// TwinCAT 3 PLC project PLCserra
// ProgramVersion: 3.1.4024.0
// libraries:
//   Tc2_Standard, * (Beckhoff Automation GmbH)
//   Tc2_System, * (Beckhoff Automation GmbH)
//   Tc3_Module, * (Beckhoff Automation GmbH)
// project tree:
//   / PlcTask.TcTTO (not stored)
//   POUs/ main.TcPOU
// real-time tasks:
//   TASK PlcTask: cycle T#10ms, priority 20, ADS port 350

// ---- POUs/main.TcPOU
PROGRAM main
VAR
	//attuatori
	AttuatBraccioGiu : BOOL := FALSE;
	AttuatBraccioSu : BOOL := FALSE;
	AttuatBraccioSx : BOOL := FALSE;
	AttuatBraccioDx : BOOL := FALSE;
	AttuatBraccioPresa : BOOL := FALSE;
	AttuatBraccioRilascio : BOOL := FALSE;
	AttuatRiempiSerbatoio : BOOL := FALSE;
	AttuatSvuotaSerbatoio : BOOL := FALSE;
	AttuatFinestra : BOOL := FALSE;
	AttuatCondizionatore : BOOL := FALSE;
	AttuatRullo : BOOL := FALSE;
	AttuatLampada : BOOL := FALSE;
	//sensori
	SensoreFCB : BOOL := FALSE;
	SensoreFCT : BOOL := FALSE;
	SensoreFCS : BOOL := FALSE;
	SensoreFCD : BOOL := FALSE;
	SensoreFineCorsaPianta2 : BOOL := FALSE;
	SensoreGrasp : BOOL := FALSE;
	SensoreRelease : BOOL := FALSE;
	SensoreRulloOccupato : BOOL := FALSE;
	SensoreVascaPienaVuota : BOOL := FALSE;
	SensoreSerbatoioOn : BOOL := FALSE;
	SensoreSerbatoioFull : BOOL := FALSE;
	SensoreSerbatoioEmpty : BOOL := FALSE;
	SensoreCondizionatore : BOOL := FALSE;
	SensoreLuci : BOOL := FALSE;
	SensoreFinestra : BOOL := FALSE;
	SensoreTempCalda : BOOL := FALSE;
	SensoreTempFredda : BOOL := FALSE;
	SensorePianta1Pronta : BOOL := FALSE;
	SensorePianta2Pronta : BOOL := FALSE;
	SensoreStart : BOOL := FALSE;
	SensoreReset : BOOL := FALSE;
	//Variabili Controllo temperatura
	TemperaturaAttuale : INT;
	TemperaturaOttimale : INT := 36;
	
	//Variabili Controllo luce
	durataGiorno : INT;
	durataNotte : INT;
	
	//Variabili controllo Serbatoio
	LivelloSerbatoio : INT;
	LivelloSerbatoioMax : INT;
	
	
	SerbatoioVuoto: BOOL;
	Pianta1Pronta: INT;
	SerbatoioPieno: BOOL;
	VascaVuota: BOOL;
	VascaPiena: BOOL;
	Pianta2Pronta: BOOL;
	RulloPieno: BOOL;
	SopraPianta1: INT;
	PrendiPianta1: BOOL;
	PosizionePianta1: BOOL;
	Pianta1Grasped: BOOL;
	Pianta1Sopra: BOOL;
	Pianta1Alzata: BOOL;
	Pianta1SopraRullo: BOOL;
	Pianta1SulRullo: INT;
	SulRullo: INT;
	Pianta1SulRulloSulRullo: BOOL;
	Pianta1Rilasciata: BOOL;
	SopraPianta2: INT;
END_VAR

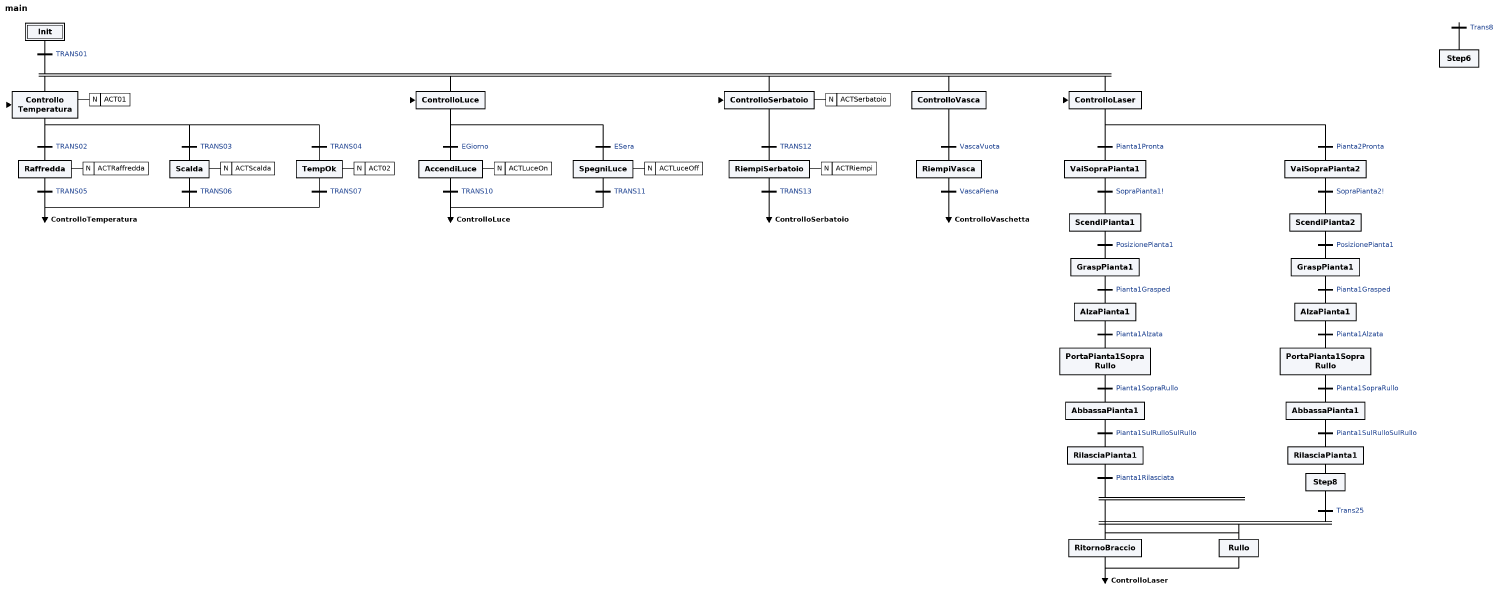
INITIAL_STEP Init:
END_STEP
TRANSITION FROM Init TO (ControlloTemperatura, ControlloLuce, ControlloSerbatoio, ControlloVasca, ControlloLaser)
    := TRANS01;
END_TRANSITION
STEP ControlloTemperatura:
    ACT01(N);
END_STEP
TRANSITION FROM ControlloTemperatura TO Raffredda
    := TRANS02;
END_TRANSITION
STEP Raffredda:
    ACTRaffredda(N);
END_STEP
TRANSITION FROM Raffredda TO ControlloTemperatura
    := TRANS05;
END_TRANSITION
TRANSITION FROM ControlloTemperatura TO Scalda
    := TRANS03;
END_TRANSITION
STEP Scalda:
    ACTScalda(N);
END_STEP
TRANSITION FROM Scalda TO ControlloTemperatura
    := TRANS06;
END_TRANSITION
TRANSITION FROM ControlloTemperatura TO TempOk
    := TRANS04;
END_TRANSITION
STEP TempOk:
    ACT02(N);
END_STEP
TRANSITION FROM TempOk TO ControlloTemperatura
    := TRANS07;
END_TRANSITION
STEP ControlloLuce:
END_STEP
TRANSITION FROM ControlloLuce TO AccendiLuce
    := EGiorno;
END_TRANSITION
STEP AccendiLuce:
    ACTLuceOn(N);
END_STEP
TRANSITION FROM AccendiLuce TO ControlloLuce
    := TRANS10;
END_TRANSITION
TRANSITION FROM ControlloLuce TO SpegniLuce
    := ESera;
END_TRANSITION
STEP SpegniLuce:
    ACTLuceOff(N);
END_STEP
TRANSITION FROM SpegniLuce TO ControlloLuce
    := TRANS11;
END_TRANSITION
STEP ControlloSerbatoio:
    ACTSerbatoio(N);
END_STEP
TRANSITION FROM ControlloSerbatoio TO RiempiSerbatoio
    := TRANS12;
END_TRANSITION
STEP RiempiSerbatoio:
    ACTRiempi(N);
END_STEP
TRANSITION FROM RiempiSerbatoio TO ControlloSerbatoio
    := TRANS13;
END_TRANSITION
STEP ControlloVasca:
END_STEP
TRANSITION FROM ControlloVasca TO RiempiVasca
    := VascaVuota;
END_TRANSITION
STEP RiempiVasca:
END_STEP
TRANSITION FROM RiempiVasca TO ControlloVaschetta
    := VascaPiena;
END_TRANSITION
STEP ControlloLaser:
END_STEP
TRANSITION FROM ControlloLaser TO VaiSopraPianta1
    := Pianta1Pronta;
END_TRANSITION
STEP VaiSopraPianta1:
END_STEP
TRANSITION FROM VaiSopraPianta1 TO ScendiPianta1
    := SopraPianta1!;
END_TRANSITION
STEP ScendiPianta1:
END_STEP
TRANSITION FROM ScendiPianta1 TO GraspPianta1
    := PosizionePianta1;
END_TRANSITION
STEP GraspPianta1:
END_STEP
TRANSITION FROM GraspPianta1 TO AlzaPianta1
    := Pianta1Grasped;
END_TRANSITION
STEP AlzaPianta1:
END_STEP
TRANSITION FROM AlzaPianta1 TO PortaPianta1SopraRullo
    := Pianta1Alzata;
END_TRANSITION
STEP PortaPianta1SopraRullo:
END_STEP
TRANSITION FROM PortaPianta1SopraRullo TO AbbassaPianta1
    := Pianta1SopraRullo;
END_TRANSITION
STEP AbbassaPianta1:
END_STEP
TRANSITION FROM AbbassaPianta1 TO RilasciaPianta1
    := Pianta1SulRulloSulRullo;
END_TRANSITION
STEP RilasciaPianta1:
END_STEP
TRANSITION FROM RilasciaPianta1 TO (RitornoBraccio, Rullo)
    := Pianta1Rilasciata;
END_TRANSITION
TRANSITION FROM ControlloLaser TO VaiSopraPianta2
    := Pianta2Pronta;
END_TRANSITION
STEP VaiSopraPianta2:
END_STEP
TRANSITION FROM VaiSopraPianta2 TO ScendiPianta2
    := SopraPianta2!;
END_TRANSITION
STEP ScendiPianta2:
END_STEP
TRANSITION FROM ScendiPianta2 TO GraspPianta1
    := PosizionePianta1;
END_TRANSITION
STEP GraspPianta1:
END_STEP
TRANSITION FROM GraspPianta1 TO AlzaPianta1
    := Pianta1Grasped;
END_TRANSITION
STEP AlzaPianta1:
END_STEP
TRANSITION FROM AlzaPianta1 TO PortaPianta1SopraRullo
    := Pianta1Alzata;
END_TRANSITION
STEP PortaPianta1SopraRullo:
END_STEP
TRANSITION FROM PortaPianta1SopraRullo TO AbbassaPianta1
    := Pianta1SopraRullo;
END_TRANSITION
STEP AbbassaPianta1:
END_STEP
TRANSITION FROM AbbassaPianta1 TO RilasciaPianta1
    := Pianta1SulRulloSulRullo;
END_TRANSITION
STEP RilasciaPianta1:
END_STEP
// no transition between RilasciaPianta1 and Step8
STEP Step8:
END_STEP
TRANSITION FROM Step8 TO (RitornoBraccio, Rullo)
    := Trans25;
END_TRANSITION
STEP RitornoBraccio:
END_STEP
// no transition between RitornoBraccio and ControlloLaser
STEP Rullo:
END_STEP
// no transition between Rullo and ControlloLaser
TRANSITION FROM ??? TO Step6
    := Trans8;
END_TRANSITION
STEP Step6:
END_STEP

ACTION ACT01:
IF TemperaturaAttuale < TemperaturaOttimale-5 THEN
	SensoreTempFredda := TRUE;
	SensoreTempCalda := FALSE;
	
ELSIF TemperaturaAttuale > TemperaturaOttimale+5 THEN
	SensoreTempCalda := TRUE;
	SensoreTempFredda := FALSE;
END_IF
END_ACTION

ACTION ACT02:
AttuatCondizionatore := FALSE;
END_ACTION

ACTION ACTLuceOff:
AttuatLampada := FALSE;
SensoreLuci := FALSE;
END_ACTION

ACTION ACTLuceOn:
AttuatLampada := TRUE;
SensoreLuci := TRUE;
END_ACTION

ACTION ACTRaffredda:
//Dovrebbe azionare il condizionare freddo
AttuatCondizionatore := TRUE;
END_ACTION

ACTION ACTRiempi:
AttuatRiempiSerbatoio := TRUE;
SensoreSerbatoioEmpty := FALSE;
END_ACTION

ACTION ACTScalda:
//Dovrebbe azionare il condizionatore caldo
AttuatCondizionatore := TRUE;
END_ACTION

ACTION ACTSerbatoio:
IF LivelloSerbatoio > 0 THEN
	IF LivelloSerbatoio = LivelloSerbatoioMax THEN
		SensoreSerbatoioFull := TRUE;
		SensoreSerbatoioEmpty := FALSE;
	END_IF
	SensoreSerbatoioEmpty := FALSE;
END_IF

IF LivelloSerbatoio = 0 THEN
	SensoreSerbatoioEmpty := TRUE;
	SensoreSerbatoioFull := FALSE;
	AttuatRiempiSerbatoio := TRUE;
END_IF
END_ACTION

TRANSITION TRANS01:
SensoreStart = TRUE AND SensoreFCTop= TRUE AND SensoreFCD = TRUE AND SensoreRulloOccupato = FALSE;
END_TRANSITION

TRANSITION TRANS02:
SensoreTempCalda := TRUE;
END_TRANSITION

TRANSITION TRANS03:
SensoreTempFredda := TRUE;
END_TRANSITION

TRANSITION TRANS04:
TemperaturaAttuale = TemperaturaOttimale;
END_TRANSITION

TRANSITION TRANS05:
AttuatCondizionatore := TRUE;
SensoreTempFredda := TRUE;
END_TRANSITION

TRANSITION TRANS06:
AttuatCondizionatore := TRUE;
END_TRANSITION

TRANSITION TRANS07:
AttuatCondizionatore := FALSE;
SensoreTempCalda := FALSE;
SensoreTempFredda := FALSE;
END_TRANSITION

TRANSITION TRANS10:
SensoreLuci := TRUE;
END_TRANSITION

TRANSITION TRANS11:
SensoreLuci := FALSE;
END_TRANSITION

TRANSITION TRANS12:
SensoreSerbatoioEmpty := TRUE;
END_TRANSITION

TRANSITION TRANS13:
SensoreSerbatoioFull := TRUE AND SensoreSerbatoioEmpty := FALSE AND AttuatRiempiSerbatoio := FALSE;
END_TRANSITION

END_PROGRAM
